FUNCTION "FC_PACKDWORD" : DWord
{ S7_Optimized_Access := 'FALSE' }
VERSION : 0.0
   VAR_INPUT
      B0 : Bool;
      B1 : Bool;
      B2 : Bool;
      B3 : Bool;
      B4 : Bool;
      B5 : Bool;
      B6 : Bool;
      B7 : Bool;
      B8 : Bool;
      B9 : Bool;
      B10 : Bool;
      B11 : Bool;
      B12 : Bool;
      B13 : Bool;
      B14 : Bool;
      B15 : Bool;
      B16 : Bool;
      B17 : Bool;
      B18 : Bool;
      B19 : Bool;
      B20 : Bool;
      B21 : Bool;
      B22 : Bool;
      B23 : Bool;
      B24 : Bool;
      B25 : Bool;
      B26 : Bool;
      B27 : Bool;
      B28 : Bool;
      B29 : Bool;
      B30 : Bool;
      B31 : Bool;
   END_VAR

   VAR_TEMP
      GW : DWord;
      INDEX : Int;
      BS : Array[0..31] of Bool;
   END_VAR


BEGIN
	;
	    #GW:=0; //GW IN TO ZERO
	    #BS[0]:=#B0;
	    #BS[1]:=#B1;
	    #BS[2]:=#B2;
	    #BS[3]:=#B3;
	    #BS[4]:=#B4;
	    #BS[5]:=#B5;
	    #BS[6]:=#B6;
	    #BS[7]:=#B7;
	    #BS[8]:=#B8;
	    #BS[9]:=#B9;
	    #BS[10]:=#B10;
	    #BS[11]:=#B11;
	    #BS[12]:=#B12;
	    #BS[13]:=#B13;
	    #BS[14]:=#B14;
	    #BS[15]:=#B15;
	    #BS[16]:=#B16;
	    #BS[17]:=#B17;
	    #BS[18]:=#B18;
	    #BS[19]:=#B19;
	    #BS[20]:=#B20;
	    #BS[21]:=#B21;
	    #BS[22]:=#B22;
	    #BS[23]:=#B23;
	    #BS[24]:=#B24;
	    #BS[25]:=#B25;
	    #BS[26]:=#B26;
	    #BS[27]:=#B27;
	    #BS[28]:=#B28;
	    #BS[29]:=#B29;
	    #BS[30]:=#B30;
	    #BS[31]:=#B31;
	    FOR #INDEX := 0 TO 31 BY 1 DO
	        IF #BS[#INDEX]THEN
	            #GW:=#GW OR (SHL(IN:=DW#16#1,N:=#INDEX));
	        END_IF;
	    END_FOR;
	        #FC_PACKDWORD := #GW; //RESULT

END_FUNCTION

FUNCTION_BLOCK "FB_ANA11"
{ S7_Optimized_Access := 'FALSE' }
VERSION : 0.0
   VAR_INPUT
      XQ11 : Int;   // Значение с поля
      XG24 : Bool;
      SFLT : Bool;
   END_VAR

   VAR_OUTPUT
      QV : Real;   // Показание датчика
      GL2 : Bool;
      GL1 : Bool;
      GL0 : Bool;
      GH0 : Bool;
      GH1 : Bool;
      GH2 : Bool;
      GVI : Bool;
      GVX : Bool;
   END_VAR

   VAR
      GVX2 : Bool;
      GVX3 : Bool;
      GVHL : Bool;
      GMW : Bool;
      GMJ : Bool;
      GVX1 : Bool;
      GMZ1 : Bool;
      GMZ2 : Bool;
      GMZ3 : Bool;
      GMZ4 : Bool;
      AVL1 : Real;
      AVH1 : Real;
      GW1 : DWord;
      X_J : Real;
      X11_J : Real;
      J_Last_Val : Real;
      PHA : Int;
      ST : Int;
      CMD : Int;
      KMJN : Bool;
      KMWN : Bool;
      ST1 : Int;
      AVJ : Real := 45.0;
      AL1 : Real := 30.0;
      AH1 : Real := 60.0;
      KMW : Bool;
      KMJ : Bool;
      AVL3 : Real;
      AVL2 : Real := 10.0;
      AVH2 : Real := 80.0;
      AVH3 : Real := 100.0;
      AVZ3 : Real := 40.0;
      KMZ : Int := 4;
      CODCBR : Real := -27648.0;
      CODL : Real;
      GIS : Real;
      GIS_GVHL : Real := 1.0;
      AL0 : Real := 35.0;
      AH0 : Real := 55.0;
      DEADZONE : Real;
   END_VAR


BEGIN


	(*Шаг 1  Установка  режимов  обработки  и  замены  параметров *)
	CASE #KMZ OF
	    1 : #GMZ1:=1; #GMZ2:=0; #GMZ3:=0; #GMZ4:=0;
	    2 : #GMZ2:=1; #GMZ1:=0; #GMZ3:=0; #GMZ4:=0;
	    3 : #GMZ3:=1; #GMZ1:=0; #GMZ2:=0; #GMZ4:=0;
	    4 : #GMZ4:=1; #GMZ1:=0; #GMZ2:=0; #GMZ3:=0;
	END_CASE;

	CASE #PHA OF
	    7:  #GMJ:=1; #KMJ:=1; #CMD:=0;  (* УСТАНОВИТЬ РЕЖИМ ИМИТАЦИИ *)
	    8:  #GMJ:=0; #KMJN:=1; #CMD:=0; (* CБРОСИТЬ РЕЖИМ ИМИТАЦИИ *)
	    9:  #GMW:=1; #KMW:=1; #CMD:=0;  (* УСТАНОВИТЬ РЕЖИМ МАСКИРОВАНИЯ *)
	    10: #GMW:=0; #KMWN:=1; #CMD:=0; (* СБРОСИТЬ РЕЖИМ МАСКИРОВАНИЯ *)
	END_CASE;
	#PHA:=0;

	(* ОБРАБОТКА АНАЛОГОВОГО СИГНАЛА *)
	//X11_J:=X11;
	#X11_J:=INT_TO_REAL((#XQ11));
	#X_J:=(#X11_J-#CODL)/(27648.0-#CODL)*(#AVH3-#AVL3)+#AVL3;
	IF (#X11_J < #CODL-#GIS_GVHL) OR (#X11_J > 27648.0+#GIS_GVHL) THEN #GVHL:=1; END_IF;
	IF (#X11_J > #CODL) & (#X11_J < 27648.0-#CODL) THEN #GVHL:=0; END_IF;
	IF NOT #GMW THEN
	    #GVX1:=#SFLT;  (*Неисправность  S 800  *)
	    #GVX2:=#XG24;   (*Неисправность датчика *)
	    #GVX3:=(NOT #XG24)&(#X11_J<=#CODCBR OR #X11_J>=32704.0); (*Обрыв, короткое замыкание*)
	END_IF;

	(* ОБРАБОТКА РЕЖИМА ИМИТАЦИИ *)
	IF #GMJ THEN
	    #QV:=#AVJ;
	    #GVX:=0;
	    #ST1:=2;   (*СТАТУС - В норме*)
	ELSE
	    IF #GMW THEN  (* ОБРАБОТКА РЕЖИМА МАСКИРОВАНИЯ *)
	        #QV:=#X_J;
	        IF (ABS(#QV)<#DEADZONE) THEN
	             #QV:=0.0;
	        END_IF;
	        #GVX:=1;
	        #ST1:=2; (*СТАТУС - В норме*)
	    ELSE
	        IF #GVX1 OR #GVX2 OR #GVX3 OR #GVHL THEN   (* ОБРАБОТКА НЕИСПРАВНОСТЕЙ И РЕЖИМОВ ЗАМЕН *)
	            #ST1:=16; (*СТАТУС - Значение не контролируется*)
	            IF #GMZ1 THEN #QV:=#AL1+(#AH1-#AL1)/2.0; END_IF;
	            IF #GMZ2 THEN #QV:=#J_Last_Val; END_IF;
	            IF #GMZ3 THEN #QV:=#AVZ3; END_IF;
	            IF #GMZ4 THEN #QV:=#X_J;
	                IF (ABS(#QV)<#DEADZONE) THEN
	                    #QV:=0.0;
	                END_IF;
	            END_IF;
	            #GVX:=1;
	        ELSE
	            #J_Last_Val:=#QV;   (* ТЕКУЩЕЕ ЗНАЧЕНИЕ АНАЛОГОВОГО ПАРАМЕТРА *)
	            #QV:=#X_J;
	            IF (ABS(#QV)<#DEADZONE) THEN
	                #QV:=0.0;
	            END_IF;
	            #GVX:=0;
	            #ST1:=2; (*СТАТУС - В норме*)
	        END_IF;
	    END_IF;
	END_IF;

	(*IF NOT GMW THEN 9_04_2006 init - Vitaliy *)
	(* ОБРАБОТКА УСТАВОК *)
	#GH0:=(((#QV>#AH0) OR #GH0&(#QV>(#AH0-#GIS)))) AND ( NOT #GMW);  (*Максимальное допустимое*)
	#GH1:=(((#QV>#AH1) OR #GH1&(#QV>(#AH1-#GIS)))) AND (NOT #GMW);   (*Максимальное предупредительное*)
	#GH2:=(((#QV>#AVH2) OR #GH2&(#QV>(#AVH2-#GIS)))) AND (NOT #GMW); (*Максимальное Аварийное*)
	#GL0:=(((#QV<#AL0) OR #GL0&(#QV<(#AL0+#GIS)))) AND ( NOT #GMW);  (*Минимальное допустимое*)
	#GL1:=(((#QV<#AL1) OR #GL1&(#QV<(#AL1+#GIS)))) AND (NOT #GMW);   (*Минимальное предупредительное*)
	#GL2:=(((#QV<#AVL2) OR #GL2&(#QV<(#AVL2+#GIS)))) AND (NOT #GMW); (*Минимальное Аварийное*)
	#GVI:=NOT(#GH0 OR #GL0 OR #GMW);

	(* ФОРМИРОВАНИЕ ТЕКУЩЕГО СТАТУСА *)
	IF NOT #GMW THEN
	    IF(#ST1<>16) THEN   (* ЕСЛИ ЗНАЧЕНИЕ КОНТРОЛИРУЕТСЯ *)
	        IF(#GH2) THEN
	        #ST1:=4;    (*СТАТУС - Значение максимальное аварийное*)
	        ELSE
	            IF(#GH1) THEN
	            #ST1:=6;  (*СТАТУС - Значение максимальное предупр*)
	            ELSE
	                IF(#GH0) THEN
	                #ST1:=8;      (*СТАТУС - Значение максимальное  допустимое*)
	                ELSE
	                    IF(#GL2) THEN
	                    #ST1:=14;      (*СТАТУС - Значение минимальное  аварийное*)
	                    ELSE
	                        IF(#GL1) THEN
	                        #ST1:=12;      (*СТАТУС - Значение минимальное предельное *)
	                        ELSE
	                            IF(#GL0) THEN
	                            #ST1:=10;      (*СТАТУС - Значение минимальное допустимое *)
	                            END_IF;
	                        END_IF;
	                    END_IF;
	                END_IF;
	            END_IF;
	        END_IF;
	    END_IF;
	END_IF;
	#ST:=#ST1;
	(* УПАКОВКА GW1 *)
	#GW1:="FC_PACKDWORD"(  B0:=#KMJ,
	        B1:=#KMJN,
	        B2:=#KMW,
	        B3:=#KMWN,
	        B4:=0,
	        B5:=0,
	        B6:=#GMJ,
	        B7:=NOT #GMJ,
	        B8:=#GMW,
	        B9:=NOT #GMW,
	        B10:=0,
	        B11:=0,
	        B12:=0,
	        B13:=0,
	        B14:=#GVX,
	        B15:=#GVX1,
	        B16:=#GVX2,
	        B17:=#GVX3,
	        B18:=#GVHL,
	        B19:=#GL2,
	        B20:=#GL1,
	        B21:=#GH1,
	        B22:=#GH2,
	        B23:=#GL0,
	        B24:=#GH0,
	        B25:=0,
	        B26:=0,
	        B27:=#GMZ1,
	        B28:=#GMZ2,
	        B29:=#GMZ3,
	        B30:=#GMZ4,
	        B31:=0);

	(* СЧЕТЧИК И СБРОС КОМАНД *)
	IF(#CMD<10 AND (#KMJ OR #KMJN OR #KMW OR #KMWN)) THEN
	    #CMD:=#CMD+1;
	ELSE
	    #KMJ:=0;
	    #KMJN:=0;
	    #KMW:=0;
	    #KMWN:=0;
	END_IF;


END_FUNCTION_BLOCK

